// TIA Portal V16 export
// export: Created 2024-05-13T12:47:23.1119358Z, ExportSetting WithDefaults, DisplayName Totally Integrated Automation Portal, DisplayVersion V16 Update 6, DisplayName TIA Portal Version Control Interface, DisplayVersion V16 Update 2, DisplayName TIA Portal Openness, DisplayVersion V16 Update 6, DisplayName TIA Portal Test Suite Advanced, DisplayVersion V16, DisplayName SINAMICS Startdrive Advanced, DisplayVersion V16 Update 5, DisplayName SINAMICS Startdrive G130, G150, S120, S150, SINAMICS MV, S210, DisplayVersion V16 Update 5, DisplayName SINAMICS Startdrive G110M, G120, G120C, G120D, G120P, G115D, DisplayVersion V16 Update 5, DisplayName STEP 7 Professional, DisplayVersion V16 Update 6, DisplayName STEP 7 Safety, DisplayVersion V16, DisplayName WinCC Advanced, DisplayVersion V16 Update 6
TYPE "SCA_Stopper"
// stored: IsFailsafeCompliant false
   STRUCT
      Status : "SCA_Status";
      IO { S7_SetPoint := 'True'} : "SCA_Stopper_IO";
      Interlock_1 { S7_SetPoint := 'True'} : "SCA_Interlock";   // Hard stopper plate
      Interlock_2 { S7_SetPoint := 'True'} : "SCA_Interlock";   // Stopper plate cushion
      Control_1 { S7_SetPoint := 'True'} : "RMP_UDT_CONTROL";   // Hard stopper plate
      Control_2 { S7_SetPoint := 'True'} : "RMP_UDT_CONTROL";   // Stopper plate cushion
      Device_name { S7_SetPoint := 'True'} : String[40];
   END_STRUCT;
END_TYPE
